(* Schneider Machine Expert - Basic project contoh 2, file version 1.7.0.0 *)
(* ProjectInformations: Name=New project *)

HARDWARE
  Cpu 0: TM221M16R/G
  EthernetConfiguration: NetworkName=M221, IpAllocationMode=FixedAddress, IpAddress=0.0.0.0, SubnetMask=0.0.0.0
  SerialLineConfiguration: Baud=Baud19200, Parity=ParityEven, DataBits=DataBits8, StopBits=StopBits1, PhysicalMedium=PhysicalMediumRs485, TransmissionMode=TransmissionModeModbusRtu, SlaveId=1, Addressing=SlaveAddressing
  MastTask: UsePeriodScanMode=false, PeriodScan=100
  FastTask: Period=255
  CpuBehavior: StartingMode=StartAsPreviousState, AutoSaveRamOnEeprom=true, WatchdogPeriod=250

SYMBOLS  (address, symbol, comment, settings)
  %I0.1       "S1"
  %I0.2       "S2"

POU New POU
  (* SectionNumber=1 *)

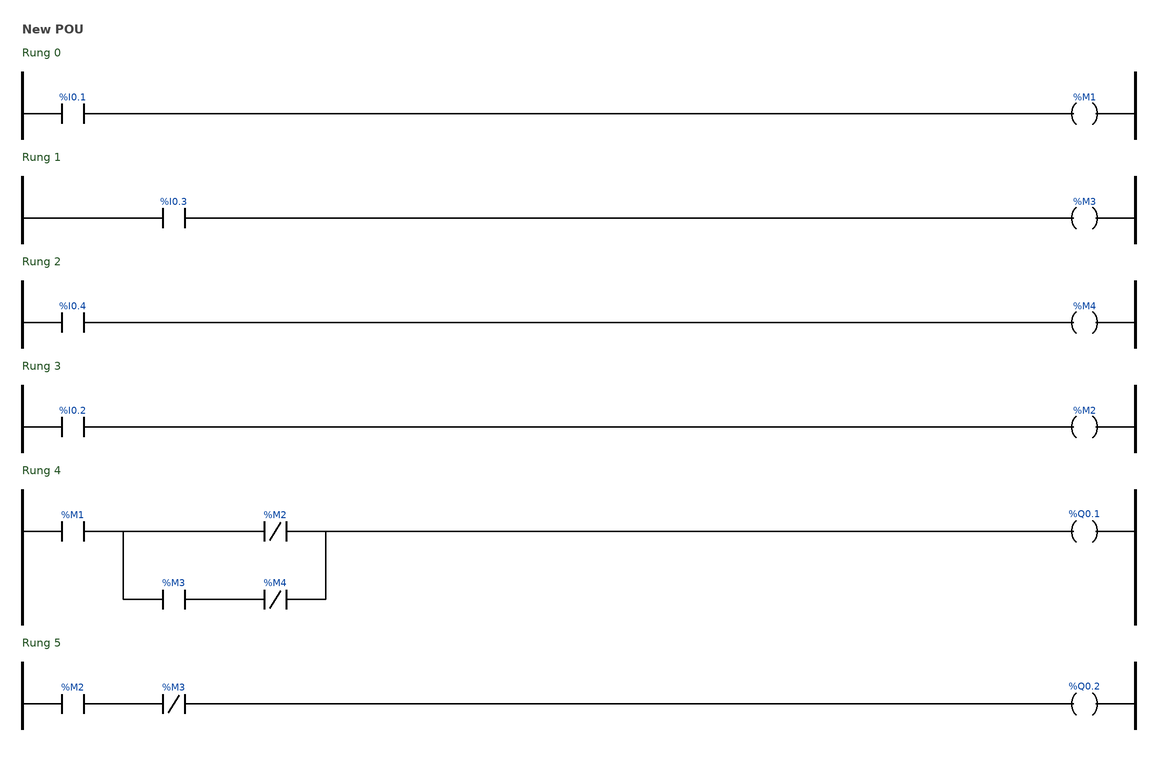

// Rung 0
  LD %I0.1
  ST %M1
  // as ST:
  //   %M1 := %I0.1;

// Rung 1
  LD %I0.3
  ST %M3
  // as ST:
  //   %M3 := %I0.3;

// Rung 2
  LD %I0.4
  ST %M4
  // as ST:
  //   %M4 := %I0.4;

// Rung 3
  LD %I0.2
  ST %M2
  // as ST:
  //   %M2 := %I0.2;

// Rung 4
  LD %M1
  AND(N %M2
  OR( %M3
  ANDN %M4
  )
  )
  ST %Q0.1
  // as ST:
  //   %Q0.1 := %M1 AND (NOT %M2 OR %M3 AND NOT %M4);

// Rung 5
  LD %M2
  ANDN %M3
  ST %Q0.2
  // as ST:
  //   %Q0.2 := %M2 AND NOT %M3;
